PROGRAM prgEHE
VAR
	fbTempH08					: FB_TempS_Ext_Input;
	fbTempH09					: FB_TempS_Ext_Input;
	fbH08_1						: FB_EHE_Linear_AO;			//{#lynus.ag#()}
	fbH08_2						: FB_EHE_Linear_AO;			//{#lynus.ag#()}
	fbH09_1						: FB_EHE_Linear_AO;			//{#lynus.ag#()}
	bSOnEmergPowerOffH08_1		: BOOL;						//{#lynus.ag#()}
	bSOnEmergPowerOffH08_2		: BOOL;						//{#lynus.ag#()}
	bSOnEmergPowerOffH09_1		: BOOL;						//{#lynus.ag#()}
	byErrorWarningH08_1			: BYTE;						//{#lynus.ag#()}
	byErrorWarningH08_2			: BYTE;						//{#lynus.ag#()}
	byErrorWarningH09_1			: BYTE;						//{#lynus.ag#()}
END_VAR
VAR PERSISTENT
	bOnEmergPowerOffH08_1		: BOOL;						//{#lynus.ag#()}
	bOnEmergPowerOffH08_2		: BOOL;						//{#lynus.ag#()}
	bOnEmergPowerOffH09_1		: BOOL;						//{#lynus.ag#()}
END_VAR

//Power Data
//each Heating Element 9kW

fbTempH08(
	bEnable:= TRUE, 
	rTemperatureOffset:= , 
	bExtErrorTemp:= prgHoneywell.fbHoneywellCntr.bErrorFunction OR prgHoneywell.fbHoneywellCntr.bErrorTemp_H08_Below OR prgHoneywell.fbHoneywellCntr.bErrorTemp_H08_Top, 
	rExtTempValue:= (prgHoneywell.fbHoneywellCntr.rBufferTemp_H08_Below + prgHoneywell.fbHoneywellCntr.rBufferTemp_H08_Top) / 2, 
	stDataTempS=> , 
	diNrOfTempS_OUT=> );
	
fbTempH09(
	bEnable:= TRUE, 
	rTemperatureOffset:= , 
	bExtErrorTemp:= prgHoneywell.fbHoneywellCntr.bErrorFunction OR prgHoneywell.fbHoneywellCntr.bErrorTemp_H09_WW, 
	rExtTempValue:= prgHoneywell.fbHoneywellCntr.rBufferTemp_H09_WW, 
	stDataTempS=> , 
	diNrOfTempS_OUT=> );

//Buffer House	
fbH08_1.stSetupEHE.bOnEmergPowerOff := bOnEmergPowerOffH08_1;
	fbH08_1.stSetupEHE.bDisableLegionellaPr := TRUE;
	
fbH08_1(
	bEnable:= , 
	bPowerDataInvers:= , 
	bNoLinear:= FALSE,
	diNrOfEMS_IN:= prgEMS.EMS.diNrOfEMS_OUT, 
	diNrOfEM_IN_EHE:= , 
	diNrOfTempS_IN:= fbTempH08.diNrOfTempS_OUT, 
	stSetupEHE:= , 
	stDataEHE=> , 
	diNrOfEHE_OUT=> , 
	rTargetPowerForExtFunc=> );	
	
byErrorWarningH08_1 := fbH08_1.stDataEHE.byErrorWarning;
	bSOnEmergPowerOffH08_1 := fbH08_1.stDataEHE.bSOnEmergPowerOff;

fbH08_2.stSetupEHE.bOnEmergPowerOff := bOnEmergPowerOffH08_2;
	fbH08_2.stSetupEHE.bDisableLegionellaPr := TRUE;
	
fbH08_2(
	bEnable:= , 
	bPowerDataInvers:= , 
	bNoLinear:= FALSE,
	diNrOfEMS_IN:= prgEMS.EMS.diNrOfEMS_OUT, 
	diNrOfEM_IN_EHE:= , 
	diNrOfTempS_IN:= fbTempH08.diNrOfTempS_OUT, 
	stSetupEHE:= , 
	stDataEHE=> , 
	diNrOfEHE_OUT=> , 
	rTargetPowerForExtFunc=> );

byErrorWarningH08_2 := fbH08_2.stDataEHE.byErrorWarning;
	bSOnEmergPowerOffH08_2 := fbH08_2.stDataEHE.bSOnEmergPowerOff;	
	
//Warmwater Boiler	
fbH09_1.stSetupEHE.bOnEmergPowerOff := bOnEmergPowerOffH09_1;

fbH09_1(
	bEnable:= , 
	bPowerDataInvers:= , 
	bNoLinear:= FALSE,
	diNrOfEMS_IN:= prgEMS.EMS.diNrOfEMS_OUT, 
	diNrOfEM_IN_EHE:= , 
	diNrOfTempS_IN:= fbTempH09.diNrOfTempS_OUT, 
	stSetupEHE:= , 
	stDataEHE=> , 
	diNrOfEHE_OUT=> , 
	rTargetPowerForExtFunc=> );
	
byErrorWarningH09_1 := fbH09_1.stDataEHE.byErrorWarning;
	bSOnEmergPowerOffH09_1 := fbH09_1.stDataEHE.bSOnEmergPowerOff;

END_PROGRAM

(* stored: Version 1.1.0.1, ProductVersion 3.1.4024.9
   POU prgEHE: Id {3eb3bd4d-209f-4c19-b404-3e1f2106f2fb}, SpecialFunc None *)
